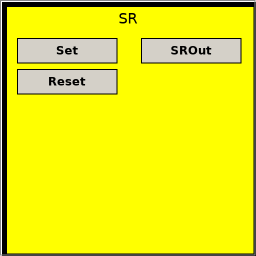
VISUALIZATION V_PH_SR  // 256x256
VAR_INPUT
	stSafetySR				:ST_SAFETY_FBSR;
END_VAR
    Rectangle (2,2 256x256), colour toggle: stSafetySR.bGeneralError
    Label (5,6 246x25), "SR"
    RoundedRectangle (17,69 100x25), "Reset", colour toggle: stSafetySR.uStatus.stStatusWords.wInputs.9
    RoundedRectangle (141,38 100x25), "SROut", colour toggle: stSafetySR.uStatus.stStatusWords.wOutputs.1
    RoundedRectangle (17,38 100x25), "Set", colour toggle: stSafetySR.uStatus.stStatusWords.wInputs.8
    Textfield (17,226 234x25), text list: 'TL_FbStateSetReset', text index: stSafetySR.eState
END_VISUALIZATION

(* stored: Version 1.1.0.1, ProductVersion 3.1.4024.4
   Visu V_PH_SR: Id {e28c5517-ea44-4a7e-944b-bda25be65705} *)
